PROGRAM MAIN
VAR
END_VAR

P_task1();

END_PROGRAM

(* stored: Version 1.1.0.1, ProductVersion 3.1.4024.12
   POU MAIN: Id {3ad56c70-386f-4f13-acfa-b11857897101}, SpecialFunc None *)
